{attribute 'enable_dynamic_creation'}
FUNCTION_BLOCK FutureMCGearIn EXTENDS FB_AbstructFuture
VAR_INPUT
END_VAR
VAR_OUTPUT
END_VAR
VAR
	_fb_gear_in	: MC_GearIn;
	_mc_reset	: MC_Reset;
	_axis_main: REFERENCE TO AXIS_REF;
	_axis_sub: REFERENCE TO AXIS_REF;
	_ratio_numerator	: MC_LREAL := 1;
	_ratio_denominator	: UINT := 1;
	_acceleration: MC_LREAL;
	_deceleration: MC_LREAL;
	_jerk		: MC_LREAL;
	_option : ST_GearInOptions;
	_buffer_mode : MC_BufferMode;
	_error_id :HRESULT;
	_exec_state : UDINT;
	_reset_state : UDINT;
END_VAR

METHOD error_reset : BOOL // Must be overrided if future has any errors.
_error_id := _fb_gear_in.ErrorID;
IF _error_id <> 0 THEN
	CASE _reset_state OF
		0:
			_mc_reset(Axis := _axis_main, Execute := FALSE);
			_mc_reset(Axis:= _axis_main, Execute := TRUE );
			_reset_state := 1;
		1:
			IF _mc_reset.Busy THEN
				_mc_reset(Axis:= _axis_main,Execute := FALSE);
			END_IF
			IF _mc_reset.Done AND NOT _mc_reset.Busy THEN
				_reset_state := 2;
			END_IF
		2:
			_mc_reset(Axis := _axis_sub, Execute := FALSE);
			_mc_reset(Axis:= _axis_sub, Execute := TRUE );
			_reset_state := 3;
		3:
			IF _mc_reset.Busy THEN
				_mc_reset(Axis:= _axis_main,Execute := FALSE);
			END_IF
			IF _mc_reset.Done AND NOT _mc_reset.Busy THEN
				_reset_state := 4;
			END_IF
		4:
			_mc_reset(Axis:= _axis_sub,Execute := FALSE);
			error_reset := TRUE;
	END_CASE
ELSE
	error_reset := TRUE;
END_IF
END_METHOD

METHOD execute : BOOL // Return TRUE if finish.
execute := FALSE;
CASE _exec_state OF
	0:
		_fb_gear_in(Master := _axis_main,Slave := _axis_sub,Execute := FALSE);
		_fb_gear_in(
			Execute := TRUE,
			Master := _axis_main,
			Slave := _axis_sub,
			RatioNumerator := _ratio_numerator,
			RatioDenominator := _ratio_denominator,
			Acceleration := _acceleration,
			Deceleration := _deceleration,
			Jerk := _jerk,
			BufferMode := _buffer_mode,
			Options := _option
		);
		_exec_state := 1;
	1:
		IF _fb_gear_in.Busy THEN
			_fb_gear_in(Master := _axis_main,Slave := _axis_sub,Execute := FALSE);
		END_IF
		IF NOT _fb_gear_in.Execute AND NOT _fb_gear_in.Busy THEN
			_exec_state := 2;
		END_IF
	2:
		IF _fb_gear_in.InGear OR _fb_gear_in.Error THEN
			_exec_state := 3;
		END_IF
	3:
		execute := TRUE;
		
END_CASE

IF _error_id = 0 AND _fb_gear_in.ErrorID <> 0 THEN
	_reset_state := 0;
END_IF

_error_id := _fb_gear_in.ErrorID;
END_METHOD

METHOD init : BOOL // Return TRUE if finish.

VAR
	axis: INT;
END_VAR
_exec_state := 0;
_reset_state := 0;
_error_id := _fb_gear_in.ErrorID;
init := TRUE;
END_METHOD

PROPERTY nErrorID : HRESULT
GET
nErrorID := _error_id;
END_GET
SET
END_SET
END_PROPERTY

METHOD set_options : BOOL
VAR_INPUT
	ratio_numerator	: MC_LREAL;
	ratio_denominator	: UINT;
	acceleration	: MC_LREAL;		// Set deceleration in case let moving axis halt.
	deceleration	: MC_LREAL;		// Set deceleration in case let moving axis halt.
	jerk			: MC_LREAL;		// Set jerk in case let moving axis halt.
	buffer_mode : MC_BufferMode;
	option : ST_GearInOptions;
END_VAR
_ratio_numerator	:= ratio_numerator;
_ratio_denominator	:= ratio_denominator;
_acceleration := acceleration;
_deceleration := deceleration;
_jerk := jerk;
_buffer_mode := buffer_mode;
_option := option;
END_METHOD

METHOD set_parameters : BOOL
VAR_INPUT
	axis_main : REFERENCE TO AXIS_REF;
	axis_sub : REFERENCE TO AXIS_REF;

END_VAR
_axis_main REF= axis_main;
_axis_sub REF= axis_sub;
END_METHOD

END_FUNCTION_BLOCK

(* stored: Version 1.1.0.1, ProductVersion 3.1.4024.15
   POU FutureMCGearIn: Id {c980d3b9-cb89-4ac9-8181-828a59352e34}, SpecialFunc None
   Method error_reset: Id {152daf12-3e4a-4bad-860e-f57ffb1137cc}
   Method execute: Id {38e13172-ea1a-4a10-9c1c-7219caa32009}
   Method init: Id {439fe697-6317-4d2e-9de0-8662a4ce5f6d}
   Property nErrorID: Id {f9a35e4f-a004-40b5-b6d3-9e868fd57c8a}
   Get Get: Id {85617870-8735-40c7-8fc0-c0a0b5d9eb30}
   Set Set: Id {487f3c0e-3427-447c-9947-c72db07345e9}
   Method set_options: Id {ed58e2fc-3f0d-48ce-8830-8d7de2e7b377}
   Method set_parameters: Id {ee4621b6-91d7-48a6-8302-d628a3f0f1ea} *)
